(* CoDeSys 2.3.9.31 project: Sample07.pro *)
(* Libraries: STANDARD.LIB 5.6.98 11:03:02 *)

(* Task configuration *)
TASK Standard (PRIORITY := 0, INTERVAL := T#10ms);
	MAIN
END_TASK

(* Data type *)
TYPE TComplexStruct :
STRUCT
	intVal : INT:=1200;
	dintArr: ARRAY[0..3] OF DINT:= 1,2,3,4;
	boolVal: BOOL := FALSE;
	byteVal: BYTE:=10;
	stringVal : STRING(5) := 'hallo';
	simpleStruct1:  TSimpleStruct;
END_STRUCT
END_TYPE

(* Data type *)
TYPE TSimpleStruct :
STRUCT
	lrealVal: 	LREAL  	:= 1.23;
	dintVal1:	DINT 	 := 120000;
END_STRUCT
END_TYPE

(* POU MAIN, ST *)
PROGRAM MAIN
VAR
	(*primitive Types*)
	Bool1:BOOL := FALSE;
	int1:INT := 30000;
	dint1:DINT:=125000;
	usint1:USINT:=200;
	real1:REAL:= 1.2;
	lreal1:LREAL:=3.5;

	(*string Types*)
	str1:STRING := 'this is a test string';
	str2:STRING(5) := 'hallo';

	(*struct Types*)
	complexStruct1 : TComplexStruct;
END_VAR
int1:=complexStruct1.intVal;
END_PROGRAM

(* POU StructTypes, ST *)
PROGRAM StructTypes
VAR
	simpleStruct1 : TSimpleStruct;

END_VAR
;
END_PROGRAM
